FUNCTION_BLOCK Robot
VAR_OUTPUT
	taskFailed : BOOL;
END_VAR
VAR
	cmd AT %Q* : TaskList; //server writes directly to this
	moveDist AT %Q* : WORD;
	
	statusReg AT %I* : UINT;
	
	rangefinderReading AT %I* : BYTE;
	
	bAtHome AT %I* : BOOL;
	bAtPos1 AT %I* : BOOL;
	bAtPos2 AT %I* : BOOL;	
	bMovedUp AT %I* : BOOL;
	bMovedDown AT %I* : BOOL;
	
	bMoving AT %I* : BOOL;
	
	timeout : TON;
	step : (IDLE, EXECUTE, FINISHED);
	done : BOOL;
END_VAR

CASE step OF
	IDLE:
		IF cmd <> TaskList.IDLE THEN
			taskFailed := FALSE;
			step := EXECUTE;
		END_IF
		
	EXECUTE: //perform task
		timeout(IN:= , PT:= T#5S, Q=> , ET=> );
		timeout.IN := TRUE;
		
		IF timeout.Q THEN
			timeout.IN := FALSE;
			taskFailed := TRUE;
			step := FINISHED;
			RETURN;
		END_IF
		
		bAtHome := statusReg = TaskList.HOME;
		bAtPos1 := statusReg = TaskList.POS1;
		bAtPos2 := statusReg = TaskList.POS2;
		bMovedUp := statusReg = TaskList.MOVE_UP;
		bMovedDown := statusReg = TaskList.MOVE_DOWN;
		
		done := statusReg = cmd;

		IF done THEN
			timeout.IN := FALSE;
			step := FINISHED;
		END_IF
	
	FINISHED: //task done, reset
		cmd := 0;
		moveDist := 0;
		step := IDLE;
END_CASE

END_FUNCTION_BLOCK

(* stored: Version 1.1.0.1, ProductVersion 3.1.4024.11
   POU Robot: Id {396ce13a-f994-4fc0-84ae-663917308fa1}, SpecialFunc None *)
